(* CoDeSys 2.3 export: OPTIMIZEDTIMER.EXP *)

(* POU OptimizedTimer, ST *)
PROGRAM OptimizedTimer
VAR
END_VAR
;
END_PROGRAM
